// TIA Portal V20 export
TYPE "LConSMC_typeSectionalDriveDiag"
// Diagnosedaten der Bahnzugregelung / Diagnostic data of the sectional drive
// stored: Access Published
   STRUCT
      typeOfAxis : Int;   // Type of axis 0: Invalid axis 1: Speed axis 2: Positioning axis 3: Synchronous axis
      referenceVelocity : LReal;   // [TO unit] Reference velocity which can be used for an external axis control (sectionalDriveConfig.axisCtrl = FALSE). Represents the maximum axis velocity at maximum line velocity
      diameterFactor : LReal;   // [%] Scaling factor for parameter "sectionalDriveDiag.referenceVelocity" which can be used for an external axis control (sectionalDriveConfig.axisCtrl = FALSE). Velocity setpoint = referenceVelocity * diameterFactor/100.0. The diameterFactor can directly be copied to the velocityOverride parameter of the TO (<TO>.Override.Velocity)
      torquePreControlDiag { S7_SetPoint := 'True'} : "LConSMC_typeTorquePrecontrolDiag";   // Diagnostic structure for torque precontrol
      technologyControllerDiag { S7_SetPoint := 'True'} : "LConSMC_typeTechnollogyControllerDiag";   // Diagnostic structure for technology controller
      webbreakDiag { S7_SetPoint := 'True'} : "LConSMC_typeWebbreakDetectDiag";   // Diagnostic structre for webbreak detection
   END_STRUCT;
END_TYPE
